PROGRAM tuning
VAR
END_VAR

END_PROGRAM

(* stored: Version 1.1.0.1, ProductVersion 3.1.4024.4
   POU tuning: Id {20c43aa5-e203-4113-bfd0-a68ab6b1422a}, SpecialFunc None *)
